Staubli VAL3: Robotscan.pjx

--- Robotscan.pjx ---
Parameters version=s7.9 stackSize=5000 millimeterUnit=true
Program file=CmdTxtReading.pgx
Program file=PositionTrigger.pgx
Program file=RobotMotion.pgx
Program file=Transmission.pgx
Program file=TxtReadRoom1.pgx
Program file=TxtReadRoom2.pgx
Program file=TxtReadRoom3.pgx
Program file=Txt_initData.pgx
Program file=WipeCacheRoom1.pgx
Program file=WipeCacheRoom2.pgx
Program file=WipeCacheRoom3.pgx
Program file=initdata.pgx
Program file=start.pgx
Program file=stop.pgx
Program file=stringtopoint.pgx
Program file=txt_PkgInit.pgx
Data file=Robotscan.dtx

--- Robotscan.dtx ---
bool bSignal
bool bTxt1
bool bTxt2
bool bTxt3
bool btrig = true
public dio fout = {link=fOut0}
public frame FrmDraw = {x=1000, y=-100, fatherId=world[0]}
mdesc mNomSpeed
num l_nInit = 1500
num nNumTotal = 5031
num nNumrecord
public num nTranC[6]
num nTxtTotal = 11
num n_sTxt
num ndelay = 258.323
public num nnnn
num ntime = 459.89
pointRx pfrmCad[1500] = {fatherId=FrmDraw[0]}
public pointRx shere = {x=16.915, y=-25.265, z=273.2, rx=-177, ry=0.5, rz=-161.069, fatherId=FrmDraw[0]}
public sio sSocketout = {link=Socket\sSocketout}
string sString[1500]
tool tTool = {fatherId=flange[0], ioLink=valve1}

--- Transmission.pgx ---
program Transmission()
  local num nByteOut[48]
  local string l_sString
begin
  nTranC[0]=shere[0].trsf.x
  nTranC[1]=shere[0].trsf.y
  nTranC[2]=shere[0].trsf.z
  nTranC[3]=shere[0].trsf.rx
  nTranC[4]=shere[0].trsf.ry
  nTranC[5]=shere[0].trsf.rz
  //toBinary(nTranC,6,"8.0b",nByteOut)
  //sioSet(sSocketout,nByteOut)

  l_sString=toString(".3",nTranC[0])+","+toString(".3",nTranC[1])+","+toString(".3",nTranC[2])+","
  l_sString=l_sString+toString(".3",nTranC[3])+","+toString(".3",nTranC[4])+","+toString(".3",nTranC[5])

  sSocketout=l_sString





end

--- TxtReadRoom2.pgx ---
program TxtReadRoom2()
  local string l_str
  local num nNumpoint
  local num ntext
  local string sTxtfile
begin
  $fileClose(0)
  $fileClose(1)
  $fileClose(2)
  $fileClose(3)
  $fileClose(4)
  $fileClose(5)
  $fileClose(6)
  $fileClose(7)
  $fileClose(8)
  $fileClose(9)


  bTxt2=false
  delay(0)
  l_str=toString("1",n_sTxt)
  sTxtfile="Disk://Robotscan/path"+l_str+".txt"
  ntext=$fileOpen(sTxtfile,"r")
  if ntext<0 or ntext>9
    popUpMsg("读取文件出错"+sTxtfile)
    return
  endIf


  for nNumpoint=500 to 999
    $fileGet(ntext,sString[nNumpoint],1)
    if sString[nNumpoint]!=""
      call stringtopoint(sString[nNumpoint],nNumpoint)
    else
    endIf
  endFor
  delay(0)

  if n_sTxt==nTxtTotal-1
    n_sTxt=0
  elseIf n_sTxt!=nTxtTotal-1
    n_sTxt=n_sTxt+1
  endIf
  nNumpoint=nNumpoint-1
  $fileClose(ntext)

  $fileClose(0)
  $fileClose(1)
  $fileClose(2)
  $fileClose(3)
  $fileClose(4)
  $fileClose(5)
  $fileClose(6)
  $fileClose(7)
  $fileClose(8)
  $fileClose(9)


end

--- TxtReadRoom3.pgx ---
program TxtReadRoom3()
  local string l_str
  local num nNumpoint
  local num ntext
  local string sTxtfile
begin

  $fileClose(0)
  $fileClose(1)
  $fileClose(2)
  $fileClose(3)
  $fileClose(4)
  $fileClose(5)
  $fileClose(6)
  $fileClose(7)
  $fileClose(8)
  $fileClose(9)


  bTxt3=false
  delay(0)
  l_str=toString("1",n_sTxt)
  sTxtfile="Disk://Robotscan/path"+l_str+".txt"
  ntext=$fileOpen(sTxtfile,"r")
  if ntext<0 or ntext>9
    popUpMsg("读取文件出错"+sTxtfile)
    return
  endIf


  for nNumpoint=1000 to 1499
    $fileGet(ntext,sString[nNumpoint],1)
    if sString[nNumpoint]!=""
      call stringtopoint(sString[nNumpoint],nNumpoint)
    else
    endIf
  endFor
  delay(0)

  if n_sTxt==nTxtTotal-1
    n_sTxt=0
  elseIf n_sTxt!=nTxtTotal-1
    n_sTxt=n_sTxt+1
  endIf
  nNumpoint=nNumpoint-1
  $fileClose(ntext)

  $fileClose(0)
  $fileClose(1)
  $fileClose(2)
  $fileClose(3)
  $fileClose(4)
  $fileClose(5)
  $fileClose(6)
  $fileClose(7)
  $fileClose(8)
  $fileClose(9)


end
